// TwinCAT 3 PLC project TcUnit
// Title: TcUnit
// Company: TcUnit
// ProjectVersion: 0.0.0.2
// ProgramVersion: 3.1.0.9
// libraries:
//   Tc2_Standard, * (Beckhoff Automation GmbH)
//   Tc2_System, * (Beckhoff Automation GmbH)
//   Tc2_Utilities, * (Beckhoff Automation GmbH)
//   Tc3_Interfaces, * (Beckhoff Automation GmbH)
//   Tc3_Module, * (Beckhoff Automation GmbH)
//   Base Interfaces,newest,System
// project tree:
//   DUTs/ MaxString.TcDUT, TypeClass.TcDUT
//   POUs/assert/ FB_Assert.TcPOU
//   POUs/mock/ PrinterMock.TcPOU
//   POUs/stringbufferoutput/ IPrinter.TcIO, StringBufferOutput.TcPOU, TestResult.TcPOU
//   POUs/test/assert/ TestAssert.TcPOU
//   POUs/test/stringbufferoutput/ TestStringBufferOutput.TcPOU
//   POUs/test/ TestMain.TcPOU
//   POUs/test/util/ TestAnyToString.TcPOU
//   POUs/util/ _any_to_string.TcPOU
//   / TestTask.TcTTO
//   Version/ Global_Version.TcGVL (not stored)

CONFIGURATION TcUnit
    RESOURCE PLC ON TwinCAT3
        TASK TestTask(INTERVAL := T#10ms, PRIORITY := 20);
        PROGRAM TestMain WITH TestTask : TestMain;
    END_RESOURCE
END_CONFIGURATION

// ---- DUTs/MaxString.TcDUT
TYPE MaxString : STRING(255); END_TYPE

// ---- DUTs/TypeClass.TcDUT
{attribute 'qualified_only'}
{attribute 'strict'}
TYPE TypeClass :
(
	TYPE_BOOL := 0,
  TYPE_BIT := 1,
  TYPE_BYTE := 2,
  TYPE_WORD := 3,
  TYPE_DWORD := 4,
  TYPE_LWORD := 5,
  TYPE_SINT := 6,
  TYPE_INT := 7,
  TYPE_DINT := 8,
  TYPE_LINT := 9,
  TYPE_USINT := 10,
  TYPE_UINT := 11,
  TYPE_UDINT := 12,
  TYPE_ULINT := 13,
  TYPE_REAL := 14,
  TYPE_LREAL := 15,
  TYPE_STRING := 16,
  TYPE_WSTRING := 17,
  TYPE_TIME := 18,
  TYPE_DATE := 19,
  TYPE_DATEANDTIME := 20,
  TYPE_TIMEOFDAY := 21,
  TYPE_POINTER := 22,
  TYPE_REFERENCE := 23,
  TYPE_SUBRANGE := 24,
  TYPE_ENUM := 25,
  TYPE_ARRAY := 26,
  TYPE_PARAMS := 27,
  TYPE_USERDEF := 28,
  TYPE_NONE := 29,
  TYPE_ANY := 30,
  TYPE_ANYBIT := 31,
  TYPE_ANYDATE := 32,
  TYPE_ANYINT := 33,
  TYPE_ANYNUM := 34,
  TYPE_ANYREAL := 35,
  TYPE_LAZY := 36,
  TYPE_LTIME := 37,
  TYPE_BITCONST := 38,
  TYPE_INTERFACE := 16#F000
);
END_TYPE

// ---- POUs/stringbufferoutput/IPrinter.TcIO
INTERFACE IPrinter

METHOD print
VAR_INPUT
END_VAR
END_METHOD

END_INTERFACE

// ---- POUs/test/TestMain.TcPOU
PROGRAM TestMain
VAR
  test_assert: TestAssert;
  test_sbo: TestStringBufferOutput;
  test_anytostring: TestAnyToString;
END_VAR

test_assert();
test_sbo();
test_anytostring();

END_PROGRAM

// ---- POUs/test/assert/TestAssert.TcPOU
FUNCTION_BLOCK TestAssert
VAR_INPUT
END_VAR
VAR_OUTPUT
END_VAR
VAR
  assert: FB_Assert('TestAssert');

  test_assert_types_bool_and_real_are_different: FB_Assert('');
  test_assert_types_int_and_int_are_not_different: FB_Assert('');
  test_assert_sizes_bool_and_int_are_different: FB_Assert('');
  test_assert_sizes_string10_and_string10_are_not_different: FB_Assert('');
END_VAR

assert.AbortAfterFail := TRUE;
CASE assert.State OF
16#0000:
  IF THIS^.types_bool_and_real_are_different() THEN
    assert.State := assert.State + 16#0010;
	END_IF
16#0010:
  IF THIS^.types_int_and_int_are_not_different() THEN
    assert.State := assert.State + 16#0010;
	END_IF
16#0020:
  IF THIS^.sizes_bool_and_int_are_different() THEN
    assert.State := assert.State + 16#0010;
	END_IF
16#0030:
  IF THIS^.sizes_string10_and_string10_are_not_different() THEN
    assert.State := assert.State + 16#0010;
	END_IF
16#FFFF:
  ;
ELSE
  assert.PrintPassed('Done');
END_CASE

METHOD sizes_bool_and_int_are_different : BOOL
VAR_INPUT
END_VAR
VAR
  expected_bool: BOOL;
  actual_int: INT;
  
  expected: BOOL;
  actual: BOOL;
END_VAR
actual := test_assert_sizes_bool_and_int_are_different.sizes_are_different(expected_bool, actual_int);
expected := TRUE;
sizes_bool_and_int_are_different := assert.AreEqualBOOL(expected, actual, 'Sizes Bool and Int are different');
END_METHOD

METHOD sizes_string10_and_string10_are_not_different : BOOL
VAR_INPUT
END_VAR
VAR
  expected_string: STRING(10);
  actual_string: STRING(10);
  
  expected: BOOL;
  actual: BOOL;
END_VAR
actual := test_assert_sizes_string10_and_string10_are_not_different.sizes_are_different(expected_string, actual_string);
expected := FALSE;
sizes_string10_and_string10_are_not_different := assert.AreEqualBOOL(expected, actual, 'Sizes String(10) and String(10) are not different');
END_METHOD

METHOD types_bool_and_real_are_different : BOOL
VAR_INPUT
END_VAR
VAR
  expected_bool: BOOL;
  actual_real: REAL;

  expected: BOOL;
  actual: BOOL;
END_VAR
actual := test_assert_types_bool_and_real_are_different.types_are_different(expected_bool, actual_real);
expected := TRUE;
types_bool_and_real_are_different := assert.AreEqualBool(expected, actual, 'Types Bool and Real are different');
END_METHOD

METHOD types_int_and_int_are_not_different : BOOL
VAR_INPUT
END_VAR
VAR
  expected_int: INT;
  actual_int: INT;

  expected: BOOL;
  actual: BOOL;
END_VAR
actual := test_assert_types_int_and_int_are_not_different.types_are_different(expected_int, actual_int);
expected := FALSE;
types_int_and_int_are_not_different := assert.AreEqualBool(expected, actual, 'Types Int and Int are not different');
END_METHOD

END_FUNCTION_BLOCK

// ---- POUs/assert/FB_Assert.TcPOU
FUNCTION_BLOCK PUBLIC FB_Assert
VAR
	bMultipleLogFlag	: BOOL;
	bAbortAfterFailFlag	: BOOL;
	bAbort				: BOOL;
	nState				: UDINT;
	sInstanceName		: STRING[255];
	sLastInstance		: STRING[255];
	sLastMessage		: STRING[255];
	nLastState			: UDINT;
END_VAR

{attribute 'monitoring':='call'}
PROPERTY PUBLIC AbortAfterFail : BOOL
SET
THIS^.bAbortAfterFailFlag := AbortAfterFail;
END_SET
END_PROPERTY

METHOD AnyTypeClassToString : STRING
VAR_INPUT
  AnyTypeClass: __SYSTEM.TYPE_CLASS;
END_VAR
CASE UDINT_TO_INT(AnyTypeClass) OF
    IBaseLibrary.TypeClass.TYPE_BOOL :
        AnyTypeClassToString := 'BOOL';
    IBaseLibrary.TypeClass.TYPE_BIT :
        AnyTypeClassToString := 'BIT';
    IBaseLibrary.TypeClass.TYPE_BYTE :
        AnyTypeClassToString := 'BYTE';
    IBaseLibrary.TypeClass.TYPE_WORD :
        AnyTypeClassToString := 'WORD';
    IBaseLibrary.TypeClass.TYPE_DWORD :
        AnyTypeClassToString := 'DWORD';
    IBaseLibrary.TypeClass.TYPE_LWORD :
        AnyTypeClassToString := 'LWORD';
    IBaseLibrary.TypeClass.TYPE_SINT :
        AnyTypeClassToString := 'SINT';
    IBaseLibrary.TypeClass.TYPE_INT :
        AnyTypeClassToString := 'INT';
    ELSE
        AnyTypeClassToString := 'UNKNOWN';
END_CASE
END_METHOD

METHOD AnyValueToHexStr : STRING(80)
VAR_INPUT
  value: ANY;
END_VAR
VAR
  i: INT;
END_VAR
FOR i:=0 TO DINT_TO_INT(value.diSize)-1 DO
  AnyValueToHexStr := CONCAT(BYTE_TO_HEXSTR(value.pValue[i], 2, FALSE), AnyValueToHexStr);
END_FOR
AnyValueToHexStr := CONCAT('0x', AnyValueToHexStr);
END_METHOD

METHOD PUBLIC AreEqualBOOL : BOOL
VAR_INPUT
	bExpected	: BOOL;
	bActual		: BOOL;
	sMessage	: STRING(80);
END_VAR
IF (bExpected <> bActual) THEN
	PrintFailed(TO_STRING(bActual), TO_STRING(bExpected), '', sMessage, 'BOOL');
	AreEqualBOOL := FALSE;
ELSE
	AreEqualBOOL := TRUE;
END_IF
END_METHOD

METHOD PUBLIC AreEqualBYTE : BOOL
VAR_INPUT
	nExpected	: BYTE;
	nActual		: BYTE;
	sMessage	: STRING(80);
END_VAR
IF (nExpected <> nActual) THEN
	PrintFailed(CONCAT('16#', DWORD_TO_HEXSTR(TO_DWORD(nActual), 8, FALSE)),
				CONCAT('16#', DWORD_TO_HEXSTR(TO_DWORD(nExpected), 8, FALSE)),
				'',
				sMessage,
				'BYTE');
	AreEqualBYTE := FALSE;
ELSE
	AreEqualBYTE := TRUE;
END_IF
END_METHOD

METHOD PUBLIC AreEqualDINT : BOOL
VAR_INPUT
	nExpected	: DINT;
	nActual		: DINT;
	sMessage	: STRING(80);
END_VAR
IF (nExpected <> nActual) THEN
	PrintFailed(TO_STRING(nActual), TO_STRING(nExpected), '', sMessage, 'DINT');
	AreEqualDINT := FALSE;
ELSE
	AreEqualDINT := TRUE;
END_IF
END_METHOD

METHOD PUBLIC AreEqualDWORD : BOOL
VAR_INPUT
	nExpected	: DWORD;
	nActual		: DWORD;
	sMessage	: STRING(80);
END_VAR
IF (nExpected <> nActual) THEN
	PrintFailed(CONCAT('16#', DWORD_TO_HEXSTR(nActual, 8, FALSE)),
				CONCAT('16#', DWORD_TO_HEXSTR(nExpected, 8, FALSE)),
				'',
				sMessage,
				'DWORD');
	AreEqualDWORD := FALSE;
ELSE
	AreEqualDWORD := TRUE;
END_IF
END_METHOD

METHOD PUBLIC AreEqualGUID : BOOL
VAR_INPUT
	stExpected	: GUID;
	stActual	: GUID;
	sMessage	: STRING(80);
END_VAR
VAR
	nIdx		: BYTE;
	bEqual		: BOOL;
END_VAR
bEqual := TRUE;
bEqual := bEqual AND stExpected.Data1 = stActual.Data1;
bEqual := bEqual AND stExpected.Data2 = stActual.Data2;
bEqual := bEqual AND stExpected.Data3 = stActual.Data3;

FOR nIdx := 0 TO 7 DO
	bEqual := bEqual AND (stExpected.Data4[nIdx] = stActual.Data4[nIdx]);
END_FOR

IF (NOT bEqual) THEN
	PrintFailed('', '', '', sMessage, 'GUID');
	AreEqualGUID := FALSE;
ELSE
	AreEqualGUID := TRUE;
END_IF
END_METHOD

METHOD PUBLIC AreEqualHRESULT : BOOL
VAR_INPUT
	hResultExp	: hResult;
	hResultAct	: hResult;
	sMessage	: STRING(80);
END_VAR
IF (hResultExp <> hResultAct) THEN
	PrintFailed(CONCAT('16#', DWORD_TO_HEXSTR(TO_DWORD(hResultAct), 8, FALSE)),
				CONCAT('16#', DWORD_TO_HEXSTR(TO_DWORD(hResultExp), 8, FALSE)),
				'',
				sMessage,
				'HRESULT');
	AreEqualHRESULT := FALSE;
ELSE
	AreEqualHRESULT := TRUE;
END_IF
END_METHOD

METHOD PUBLIC AreEqualINT : BOOL
VAR_INPUT
	nExpected	: INT;
	nActual		: INT;
	sMessage	: STRING(80);
END_VAR
IF (nExpected <> nActual) THEN
	PrintFailed(TO_STRING(nActual), TO_STRING(nExpected), '', sMessage, 'INT');
	AreEqualINT := FALSE;
ELSE
	AreEqualINT := TRUE;
END_IF
END_METHOD

METHOD PUBLIC AreEqualLINT : BOOL
VAR_INPUT
	nExpected	: LINT;
	nActual		: LINT;
	sMessage	: STRING(80);
END_VAR
IF (nExpected <> nActual) THEN
	PrintFailed(TO_STRING(nActual), TO_STRING(nExpected), '', sMessage, 'LINT');
	AreEqualLINT := FALSE;
ELSE
	AreEqualLINT := TRUE;
END_IF
END_METHOD

METHOD PUBLIC AreEqualLREAL : BOOL
VAR_INPUT
	fExpected	: LREAL;
	fActual		: LREAL;
	fTolerance	: LREAL;
	sMessage	: STRING(80);
END_VAR
VAR
	fbFormatActual		: FB_FormatString;
	fbFormatExpected	: FB_FormatString;
	sFormatOption		: STRING(20);
END_VAR
IF (ABS(fExpected-fActual) > fTolerance) THEN
	IF (fTolerance >= 0.1) THEN
		sFormatOption := '%4.1F';
	ELSIF (fTolerance >= 0.01) THEN
		sFormatOption := '%4.2F';
	ELSIF (fTolerance >= 0.001) THEN
		sFormatOption := '%4.3F';
	ELSIF (fTolerance >= 0.000001) THEN
		sFormatOption := '%4.6F';
	ELSE
		sFormatOption := '%4.9F';
	END_IF

	fbFormatActual(sFormat := sFormatOption, arg1 := F_LREAL(fActual));
	fbFormatExpected(sFormat := sFormatOption, arg1 := F_LREAL(fExpected));

	PrintFailed(fbFormatActual.sOut, fbFormatExpected.sOut, TO_STRING(fTolerance), sMessage, 'LREAL');
	AreEqualLREAL := FALSE;
ELSE
	AreEqualLREAL := TRUE;
END_IF
END_METHOD

METHOD PUBLIC AreEqualLTIME : BOOL
VAR_INPUT
	tExpected		: LTIME;
	tActual			: LTIME;
	tTolerance		: LTIME;
	sMessage		: STRING(80);
END_VAR
IF (tActual < (tExpected - tTolerance)) OR (tActual > (tExpected + tTolerance)) THEN
	PrintFailed(TO_STRING(tActual), TO_STRING(tExpected), TO_STRING(tTolerance), sMessage, 'LTIME');
	AreEqualLTIME := FALSE;
ELSE
	AreEqualLTIME := TRUE;
END_IF
END_METHOD

METHOD PUBLIC AreEqualLWORD : BOOL
VAR_INPUT
	nExpected	: LWORD;
	nActual		: LWORD;
	sMessage	: STRING(80);
END_VAR
IF (nExpected <> nActual) THEN
	PrintFailed(CONCAT('16#', LWORD_TO_HEXSTR(nActual, 16, FALSE)),
				CONCAT('16#', LWORD_TO_HEXSTR(nExpected, 16, FALSE)),
				'',
				sMessage,
				'LWORD');
	AreEqualLWORD := FALSE;
ELSE
	AreEqualLWORD := TRUE;
END_IF
END_METHOD

METHOD PUBLIC AreEqualMEM : BOOL
VAR_INPUT
	pExpected	: PVOID;
	pActual		: PVOID;
	nSize		: UDINT;
	sMessage	: STRING(80);
END_VAR
IF (MEMCMP(pExpected, pActual, nSize) <> 0) THEN
	PrintFailed('', '', '', sMessage, 'MEM');
	AreEqualMEM := FALSE;
ELSE
	AreEqualMEM := TRUE;
END_IF
END_METHOD

METHOD PUBLIC AreEqualREAL : BOOL
VAR_INPUT
	fExpected	: REAL;
	fActual		: REAL;
	fTolerance	: REAL;
	sMessage	: STRING(80);
END_VAR
VAR
	fbFormatActual		: FB_FormatString;
	fbFormatExpected	: FB_FormatString;
	sFormatOption		: STRING(20);
END_VAR
IF (ABS(fExpected-fActual) > fTolerance) THEN
	IF (fTolerance >= 0.1) THEN
		sFormatOption := '%4.1F';
	ELSIF (fTolerance >= 0.01) THEN
		sFormatOption := '%4.2F';
	ELSIF (fTolerance >= 0.001) THEN
		sFormatOption := '%4.3F';
	ELSIF (fTolerance >= 0.000001) THEN
		sFormatOption := '%4.6F';
	ELSE
		sFormatOption := '%4.9F';
	END_IF

	fbFormatActual(sFormat := sFormatOption, arg1 := F_Real(fActual));
	fbFormatExpected(sFormat := sFormatOption, arg1 := F_Real(fExpected));

	PrintFailed(fbFormatActual.sOut, fbFormatExpected.sOut, TO_STRING(fTolerance), sMessage, 'REAL');
	AreEqualREAL := FALSE;
ELSE
	AreEqualREAL := TRUE;
END_IF
END_METHOD

METHOD PUBLIC AreEqualSINT : BOOL
VAR_INPUT
	nExpected	: SINT;
	nActual		: SINT;
	sMessage	: STRING(80);
END_VAR
IF (nExpected <> nActual) THEN
	PrintFailed(TO_STRING(nActual), TO_STRING(nExpected), '', sMessage, 'SINT');
	AreEqualSINT := FALSE;
ELSE
	AreEqualSINT := TRUE;
END_IF
END_METHOD

METHOD PUBLIC AreEqualSTRING : BOOL
VAR_INPUT
	sExpected	: STRING(255);
	sActual		: STRING(255);
	sMessage	: STRING(80);
END_VAR
IF (sExpected <> sActual) THEN
	PrintFailed(sActual, sExpected, '', sMessage, 'STRING');
	AreEqualSTRING := FALSE;
ELSE
	AreEqualSTRING := TRUE;
END_IF
END_METHOD

METHOD PUBLIC AreEqualTIME : BOOL
VAR_INPUT
	tExpected		: TIME;
	tActual			: TIME;
	tTolerance		: TIME;
	sMessage		: STRING(80);
END_VAR
IF (tActual < (tExpected - tTolerance)) OR (tActual > (tExpected + tTolerance)) THEN
	PrintFailed(TO_STRING(tActual), TO_STRING(tExpected), TO_STRING(tTolerance), sMessage, 'TIME');
	AreEqualTIME := FALSE;
ELSE
	AreEqualTIME := TRUE;
END_IF
END_METHOD

METHOD PUBLIC AreEqualUDINT : BOOL
VAR_INPUT
	nExpected	: UDINT;
	nActual		: UDINT;
	sMessage	: STRING(80);
END_VAR
IF (nExpected <> nActual) THEN
	PrintFailed(TO_STRING(nActual), TO_STRING(nExpected), '', sMessage, 'UDINT');
	AreEqualUDINT := FALSE;
ELSE
	AreEqualUDINT := TRUE;
END_IF
END_METHOD

METHOD PUBLIC AreEqualUINT : BOOL
VAR_INPUT
	nExpected	: UINT;
	nActual		: UINT;
	sMessage	: STRING(80);
END_VAR
IF (nExpected <> nActual) THEN
	PrintFailed(TO_STRING(nActual), TO_STRING(nExpected), '', sMessage, 'UINT');
	AreEqualUINT := FALSE;
ELSE
	AreEqualUINT := TRUE;
END_IF
END_METHOD

METHOD PUBLIC AreEqualULINT : BOOL
VAR_INPUT
	nExpected	: ULINT;
	nActual		: ULINT;
	sMessage	: STRING(80);
END_VAR
IF (nExpected <> nActual) THEN
	PrintFailed(TO_STRING(nActual), TO_STRING(nExpected), '', sMessage, 'ULINT');
	AreEqualULINT := FALSE;
ELSE
	AreEqualULINT := TRUE;
END_IF
END_METHOD

METHOD PUBLIC AreEqualUSINT : BOOL
VAR_INPUT
	nExpected	: USINT;
	nActual		: USINT;
	sMessage	: STRING(80);
END_VAR
IF (nExpected <> nActual) THEN
	PrintFailed(TO_STRING(nActual), TO_STRING(nExpected), '', sMessage, 'USINT');
	AreEqualUSINT := FALSE;
ELSE
	AreEqualUSINT := TRUE;
END_IF
END_METHOD

METHOD PUBLIC AreEqualWORD : BOOL
VAR_INPUT
	nExpected	: WORD;
	nActual		: WORD;
	sMessage	: STRING(80);
END_VAR
IF (nExpected <> nActual) THEN
	PrintFailed(CONCAT('16#', DWORD_TO_HEXSTR(TO_DWORD(nActual), 8, FALSE)),
				CONCAT('16#', DWORD_TO_HEXSTR(TO_DWORD(nExpected), 8, FALSE)),
				'',
				sMessage,
				'WORD');
	AreEqualWORD := FALSE;
ELSE
	AreEqualWORD := TRUE;
END_IF
END_METHOD

METHOD CHECK_TRUE : BOOL
VAR_INPUT
  actual: BOOL;
  message: STRING(80);
END_VAR
//CHECK_TRUE := TRUE;
END_METHOD

METHOD equal : BOOL
VAR_INPUT
  expected: ANY;
  actual: ANY;
  message: STRING(80);
END_VAR
VAR
  i: INT;
  expected_value_str: STRING(80);
  actual_value_str: STRING(80);
END_VAR
equal := FALSE;
IF expected.TypeClass <> actual.TypeClass THEN
  PrintFailed(
    TO_STRING(actual.TypeClass), 
    TO_STRING(expected.TypeClass), 
    '',
    CONCAT(message, ' Types do not match'), 
    AnyTypeClassToString(expected.TypeClass));
  RETURN;
END_IF
 
// TODO: check for strings if the size is the length size or declared size
IF (expected.diSize <> actual.diSize) THEN
  PrintFailed(
    TO_STRING(actual.diSize), 
    TO_STRING(expected.diSize), 
    '', 
    CONCAT(message, ' Typesizes do not match'), 
    AnyTypeClassToString(expected.TypeClass));
  RETURN;
END_IF
 
// Compare each byte in the ANY-types
FOR i := 0 TO DINT_TO_INT(expected.diSize)-1 BY 1 DO
    IF expected.pValue[i] <> actual.pValue[i] THEN
      // TODO: write a Function for printing the values of the type
      PrintFailed(
        AnyValueToHexStr(actual), 
        AnyValueToHexStr(expected), 
        '', 
        message, 
        AnyTypeClassToString(expected.TypeClass));
      RETURN;
    END_IF
END_FOR
equal := TRUE;
PrintPassed(message);
END_METHOD

METHOD FB_init : BOOL
VAR_INPUT
	bInitRetains : BOOL; // if TRUE, the retain variables are initialized (warm start / cold start)
	bInCopyCode : BOOL;  // if TRUE, the instance afterwards gets moved into the copy code (online change)
	sInstanceName : STRING(255);
END_VAR
THIS^.sInstanceName := sInstanceName;
END_METHOD

METHOD PUBLIC IsFalse : BOOL
VAR_INPUT
	bCondition	: BOOL;
	sMessage	: STRING(80);
END_VAR
IF bCondition THEN
	PrintFailed(BOOL_TO_STRING(bCondition), 'FALSE', '', sMessage, 'BOOL');
	IsFalse := FALSE;
ELSE
	IsFalse := TRUE;
END_IF
END_METHOD

METHOD PUBLIC IsTrue : BOOL
VAR_INPUT
	bCondition	: BOOL;
	sMessage	: STRING(80);
END_VAR
IF (NOT bCondition) THEN
	PrintFailed(TO_STRING(bCondition), 'TRUE', '', sMessage, 'BOOL');
	IsTrue := FALSE;
ELSE
	IsTrue := TRUE;
END_IF
END_METHOD

{attribute 'monitoring':='call'}
PROPERTY PUBLIC MultipleLog : BOOL
SET
THIS^.bMultipleLogFlag := MultipleLog;
END_SET
END_PROPERTY

METHOD PUBLIC PrintFailed
VAR_INPUT
	sActual		: STRING(80);
	sExpected	: STRING(80);
	sTolerance	: STRING(80);
	sMessage	: STRING(80);
	sType		: STRING(20);
END_VAR
VAR
	sState		: STRING(10);
	sString		: STRING(255);
END_VAR
IF ((THIS^.sLastMessage <> sMessage) OR (THIS^.nLastState <> THIS^.nState) OR THIS^.bMultipleLogFlag) THEN
	THIS^.sLastInstance := THIS^.sInstanceName;
	THIS^.sLastMessage := sMessage;
	THIS^.nLastState := THIS^.nState;
	
	sString := THIS^.sInstanceName;

	sState := DWORD_TO_HEXSTR(TO_DWORD(THIS^.nState), 4, FALSE);
	
	sString := CONCAT(sString, '; State: 16#');
	sString := CONCAT(sString, sState);
	
	IF (LEN(sType) > 0) THEN
		sString := CONCAT(sString, '; ');
		sString := CONCAT(sString, sType);
	END_IF
	
	IF (LEN(sMessage) > 0) THEN
		sString := CONCAT(sString, '; ');
		sString := CONCAT(sString, sMessage);
	END_IF
	
	IF (LEN(sActual) > 0) THEN
		sString := CONCAT(sString, '; Act: ');
		sString := CONCAT(sString, sActual);
	END_IF
	
	IF (LEN(sExpected) > 0) THEN
		sString := CONCAT(sString, '; Exp: ');
		sString := CONCAT(sString, sExpected);
	END_IF
	
	IF (LEN(sTolerance) > 0) THEN
		sString := CONCAT(sString, '; Tol: ');
		sString := CONCAT(sString, sTolerance);
	END_IF
	
	ADSLOGSTR(msgCtrlMask := ADSLOG_MSGTYPE_ERROR, msgFmtStr := 'Failed: %s', strArg := sString);					
				
	IF (THIS^.bAbortAfterFailFlag) THEN
		THIS^.bAbort := TRUE;
	END_IF
END_IF
END_METHOD

METHOD PUBLIC PrintPassed
VAR_INPUT
	sMessage	: STRING(80);
END_VAR
VAR
	sState		: STRING(10);
	sString		: STRING(255);	
END_VAR
IF ((THIS^.sLastMessage <> sMessage) OR (THIS^.nLastState <> THIS^.nState) OR THIS^.bMultipleLogFlag) THEN
	THIS^.sLastInstance := THIS^.sInstanceName;
	THIS^.sLastMessage := sMessage;
	THIS^.nLastState := THIS^.nState;
	
	sString := THIS^.sInstanceName;

	sState := DWORD_TO_HEXSTR(TO_DWORD(THIS^.nState), 4, FALSE);
	
	sString := CONCAT(sString, '; State: 16#');
	sString := CONCAT(sString, sState);
		
	IF (LEN(sMessage) > 0) THEN
		sString := CONCAT(sString, '; ');
		sString := CONCAT(sString, sMessage);
	END_IF
		
	ADSLOGSTR(msgCtrlMask := ADSLOG_MSGTYPE_WARN, msgFmtStr := 'Passed: %s', strArg := sString);
END_IF
END_METHOD

METHOD sizes_are_different : BOOL
VAR_INPUT
  expected: ANY;
  actual: ANY;
END_VAR
sizes_are_different := expected.diSize <> actual.diSize;
END_METHOD

PROPERTY PUBLIC State : UDINT
GET
State := THIS^.nState;
END_GET
SET
IF (THIS^.bAbort) THEN
	THIS^.nState := 16#FFFF;
ELSE
	THIS^.nState := LIMIT(0, State, 16#FFFF);
END_IF
END_SET
END_PROPERTY

METHOD PUBLIC StateMachineError : BOOL
PrintFailed('', '', '', 'Invalid State!', 'StateMachine');
THIS^.nState := 16#FFFF;
END_METHOD

METHOD types_are_different : BOOL
VAR_INPUT
  expected: ANY;
  actual: ANY;
END_VAR
types_are_different := expected.TypeClass <> actual.TypeClass;
END_METHOD

END_FUNCTION_BLOCK

// ---- POUs/test/stringbufferoutput/TestStringBufferOutput.TcPOU
FUNCTION_BLOCK TestStringBufferOutput
VAR_INPUT
END_VAR
VAR_OUTPUT
END_VAR
VAR
  assert: FB_Assert('TestStringBufferOutput');
  
  test_sbo_compose_one_message: StringBufferOutput;
  test_sbo_compose_multiple_messages: StringBufferOutput;
  test_sbo_compose_int_message: StringBufferOutput;
  test_sbo_compose_mixed_messages: StringBufferOutput;
END_VAR

assert.AbortAfterFail := TRUE;
CASE assert.State OF
16#0000:
  IF THIS^.compose_one_message() THEN
    assert.State := assert.State + 16#0010;
	END_IF
16#0010:
  IF THIS^.compose_multiple_messages() THEN
    assert.State := assert.State + 16#0010;
	END_IF
16#0020:
  IF THIS^.compose_int_message() THEN
    assert.State := assert.State + 16#0010;
	END_IF
16#0030:
  IF THIS^.compose_mixed_messages() THEN
    assert.State := assert.State + 16#0010;
	END_IF
16#FFFF:
  ;
ELSE
  assert.PrintPassed('Done');
END_CASE

METHOD compose_int_message : BOOL
VAR_INPUT
END_VAR
VAR
  expected: STRING(10);
  actual: STRING(10);
  
  expected_int: INT;
END_VAR
expected_int := 256;
test_sbo_compose_int_message.compose_message(expected_int);
expected := '256';
actual := test_sbo_compose_int_message.get_output();
compose_int_message := assert.AreEqualSTRING(expected, actual, 'Compose Int message');
END_METHOD

METHOD compose_mixed_messages : BOOL
VAR_INPUT
END_VAR
VAR
  expected: STRING(80);
  actual: STRING(80);
  
  expected_str: STRING(80);
  expected_real: REAL;
  expected_int: INT;
END_VAR
expected_str := 'foo ';
test_sbo_compose_mixed_messages.compose_message(expected_str);
expected_int := -17;
test_sbo_compose_mixed_messages.compose_message(expected_int);
expected_str := ' bar ';
test_sbo_compose_mixed_messages.compose_message(expected_str);
expected_real := 0.1;
test_sbo_compose_mixed_messages.compose_message(expected_real);
expected := 'foo -17 bar 0.1';
actual := test_sbo_compose_mixed_messages.get_output();
compose_mixed_messages := assert.AreEqualSTRING(expected, actual, 'Compose mixed messages');
END_METHOD

METHOD compose_multiple_messages : BOOL
VAR_INPUT
END_VAR
VAR
  expected: STRING(80);
  actual: STRING(80);
  
  expected_str: STRING(80);
END_VAR
expected_str := 'world';
test_sbo_compose_multiple_messages.compose_message(expected_str);
expected_str := 'hello';
test_sbo_compose_multiple_messages.compose_message(expected_str);
expected_str := 'twincat';
test_sbo_compose_multiple_messages.compose_message(expected_str);
expected := 'worldhellotwincat';
actual := test_sbo_compose_multiple_messages.get_output();
compose_multiple_messages := assert.AreEqualSTRING(expected, actual, 'Compose multiple messages');
END_METHOD

METHOD compose_one_message: BOOL
VAR_INPUT
END_VAR
VAR
  expected: STRING(80);
  actual: STRING(80);
  
  expected_str: STRING(80);
END_VAR
expected := 'hello';
test_sbo_compose_one_message.compose_message(expected);
actual := test_sbo_compose_one_message.get_output();
compose_one_message := assert.AreEqualSTRING(expected, actual, 'Compose one message');
END_METHOD

END_FUNCTION_BLOCK

// ---- POUs/stringbufferoutput/StringBufferOutput.TcPOU
FUNCTION_BLOCK StringBufferOutput
VAR_INPUT
END_VAR
VAR_OUTPUT
END_VAR
VAR
  output_message: STRING(255);
END_VAR

METHOD compose_message
VAR_INPUT
  message: ANY;
END_VAR
VAR
  message_str: MaxString;
END_VAR
message_str := _any_to_string(message);
output_message := CONCAT(output_message, message_str);
END_METHOD

METHOD get_output : STRING(255)
get_output := output_message;
END_METHOD

END_FUNCTION_BLOCK

// ---- POUs/util/_any_to_string.TcPOU
FUNCTION _any_to_string : MaxString
VAR_INPUT
  to_transform: ANY;
END_VAR
VAR
  int_ptr: POINTER TO INT;
  real_ptr: POINTER TO REAL;
  string_ptr: POINTER TO STRING;
END_VAR

CASE UDINT_TO_INT(to_transform.TypeClass) OF
TypeClass.TYPE_INT:
  int_ptr := to_transform.pValue;
  _any_to_string := TO_STRING(int_ptr^);
TypeClass.TYPE_REAL:
  real_ptr := to_transform.pValue;
  _any_to_string := TO_STRING(real_ptr^);
TypeClass.TYPE_STRING:
  string_ptr := to_transform.pValue;
  _any_to_string := string_ptr^;
ELSE
  _any_to_string := '';
END_CASE

END_FUNCTION

// ---- POUs/test/util/TestAnyToString.TcPOU
FUNCTION_BLOCK TestAnyToString
VAR_INPUT
END_VAR
VAR_OUTPUT
END_VAR
VAR
  assert: FB_Assert('TestAnyToString');
END_VAR

assert.AbortAfterFail := TRUE;
CASE assert.State OF
16#0000:
  IF THIS^.transform_int_to_string() THEN
    assert.State := assert.State + 16#0010;
	END_IF
16#0010:
  IF THIS^.transform_real_to_string() THEN
    assert.State := assert.State + 16#0010;
	END_IF
16#0020:
  IF THIS^.transform_string_to_string() THEN
    assert.State := assert.State + 16#0010;
	END_IF
16#FFFF:
  ;
ELSE
  assert.PrintPassed('Done');
END_CASE

METHOD transform_int_to_string : BOOL
VAR_INPUT
END_VAR
VAR
  expected: STRING(10);
  actual: STRING(10);
  
  expected_int: INT;
END_VAR
expected_int := 300;
actual := _any_to_string(expected_int);
expected := '300';
transform_int_to_string := assert.AreEqualSTRING(expected, actual, 'Transform Int to String');
END_METHOD

METHOD transform_real_to_string : BOOL
VAR_INPUT
END_VAR
VAR
  expected: STRING(10);
  actual: STRING(10);
  
  expected_real: REAL;
END_VAR
expected_real := 123.456;
actual := _any_to_string(expected_real);
expected := '123.456';
transform_real_to_string := assert.AreEqualSTRING(expected, actual, 'Transform Real to String');
END_METHOD

METHOD transform_string_to_string : BOOL
VAR_INPUT
END_VAR
VAR
  expected: STRING(10);
  actual: STRING(10);
END_VAR
expected := 'foobar';
actual := _any_to_string(expected);
transform_string_to_string := assert.AreEqualSTRING(expected, actual, 'Transform String to String');
END_METHOD

END_FUNCTION_BLOCK

// ---- POUs/mock/PrinterMock.TcPOU
FUNCTION_BLOCK PrinterMock IMPLEMENTS IPrinter
VAR_INPUT
END_VAR
VAR_OUTPUT
END_VAR
VAR
END_VAR

METHOD get_output : STRING(255)
VAR_INPUT
END_VAR
END_METHOD

{warning 'add method implementation'}
METHOD print
END_METHOD

END_FUNCTION_BLOCK

// ---- POUs/stringbufferoutput/TestResult.TcPOU
FUNCTION_BLOCK TestResult
VAR_INPUT
END_VAR
VAR_OUTPUT
END_VAR
VAR
  printer: IStringBufferOutput;
END_VAR

METHOD FB_init : BOOL
VAR_INPUT
	bInitRetains : BOOL; // if TRUE, the retain variables are initialized (warm start / cold start)
	bInCopyCode : BOOL;  // if TRUE, the instance afterwards gets moved into the copy code (online change)
  printer: IStringBufferOutput;
END_VAR
THIS^.printer := printer;
END_METHOD

END_FUNCTION_BLOCK
